RoboDK station: Estacion_Lab_6_0.rdk

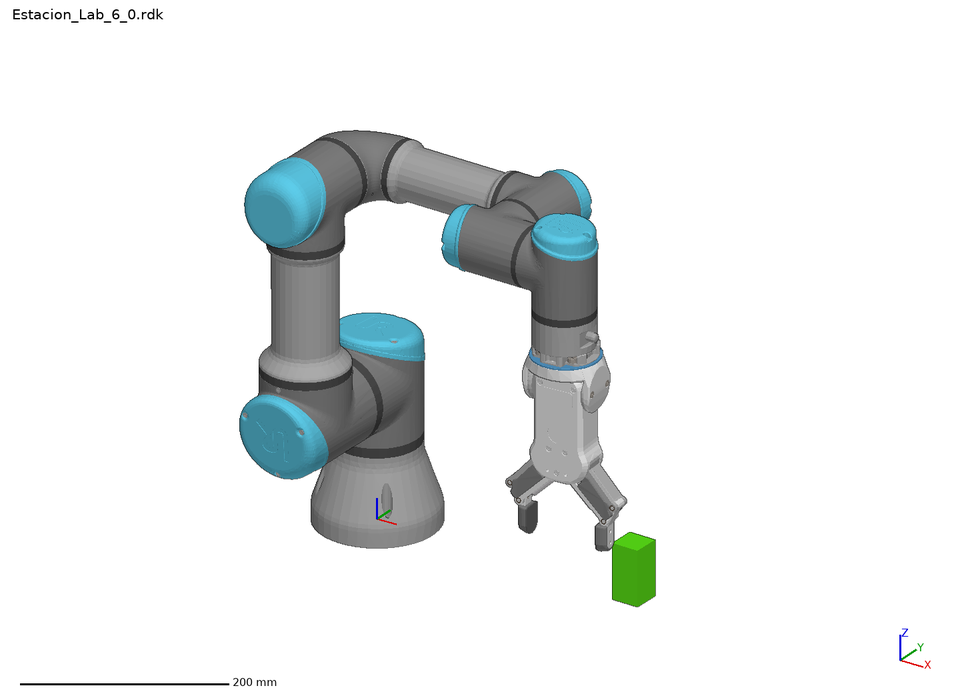
[picture v0: the station drawn from its stored meshes, robots at their saved joint values, targets as dots, program paths as lines]
Station Estacion_Lab_6_0 (saved by RoboDK 5.2.3). Poses are relative to the parent item; angles as X-Y-Z fixed-axis rotations.
  - frame UR3 Base at (0, 0, 0) mm
    - robot UR3: 6 axes, payload 3 kg, reach 500 mm, repeatability 0.1 mm, weight 11 kg
        modified DH rows (alpha deg, a mm, theta deg, d mm): 0, 0, 0, 151.9; 90, 0, 180, 0; 0, 243.65, 0, 0; 0, 213, 0, 110.4; -90, 0, 0, 83.4; 90, 0, 180, 82.4
        joint limits [-360, -360, -360, -360, -360, -360] to [360, 360, 360, 360, 360, 360]; home [0, -90, -90, 0, 90, 0]; saved at [0, -89.954, -89.954, -89.954, 89.954, 0]
      - tool RG2_v2, TCP at (0, 0, 190) mm, size 211.8 x 123.1 x 75.3 mm, geometry from RG2_v2.STEP
  - object prisma_3 at (300, 0, 0) mm, size 30 x 30 x 60 mm, geometry from prisma_2.stl
